PROGRAM TSCS_Bridge_Outputs
(*Outputs from TDU PLC to TSCS PLC*)
VAR
	// Function Blocks
	fb_Bridge_Outputs_Real_0 : FB_Bridge_Outputs_Real; // Interface for TDU real outputs
	
	// Signal Conversions
	rActPos : REAL; // Rotation system - Actual Position [deg]
	rActVel : REAL; // Rotation system - Actual Velocity [rpm]
	rSetVelRaw : REAL; //Rotation system - Velocity setpoint raw [rpm] 
	
END_VAR

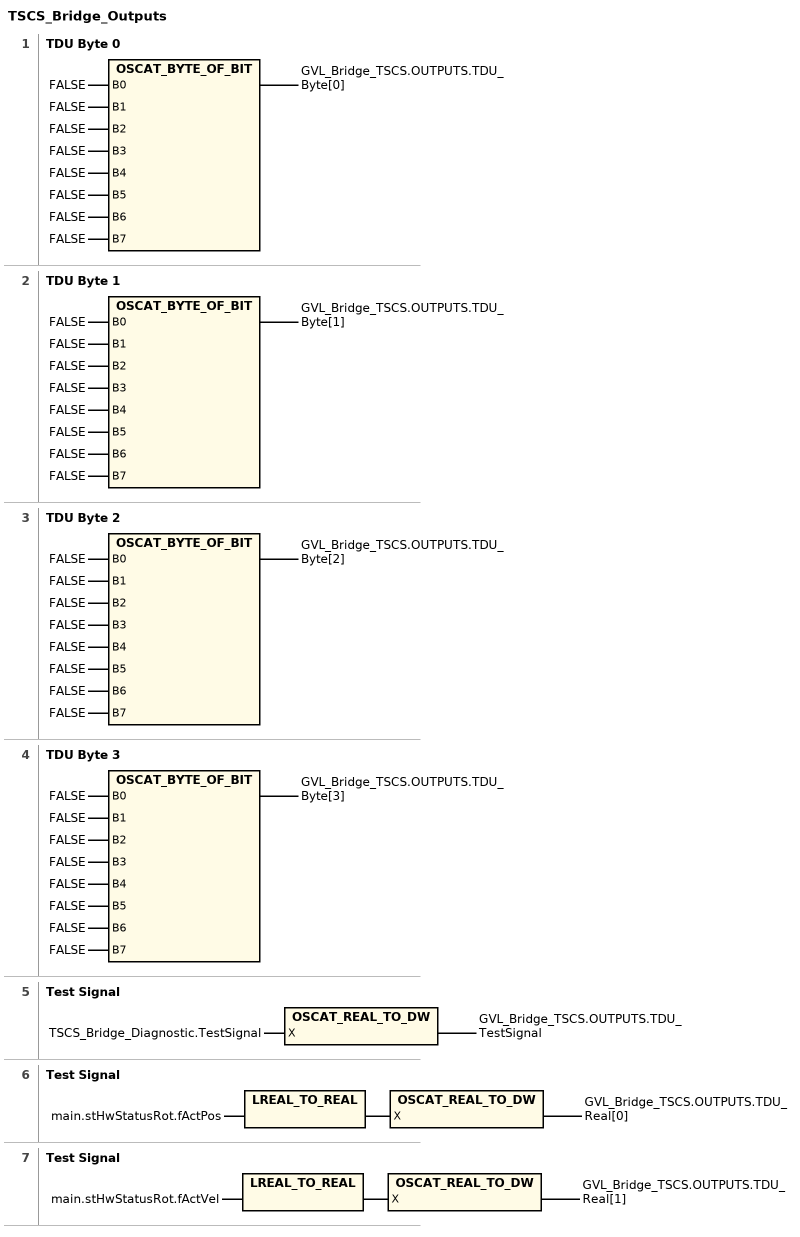
// NETWORK 1: TDU Byte 0
GVL_Bridge_TSCS.OUTPUTS.TDU_Byte[0] := OSCAT_BYTE_OF_BIT(B0 := FALSE, B1 := FALSE, B2 := FALSE, B3 := FALSE, B4 := FALSE, B5 := FALSE, B6 := FALSE, B7 := FALSE);

// NETWORK 2: TDU Byte 1
GVL_Bridge_TSCS.OUTPUTS.TDU_Byte[1] := OSCAT_BYTE_OF_BIT(B0 := FALSE, B1 := FALSE, B2 := FALSE, B3 := FALSE, B4 := FALSE, B5 := FALSE, B6 := FALSE, B7 := FALSE);

// NETWORK 3: TDU Byte 2
GVL_Bridge_TSCS.OUTPUTS.TDU_Byte[2] := OSCAT_BYTE_OF_BIT(B0 := FALSE, B1 := FALSE, B2 := FALSE, B3 := FALSE, B4 := FALSE, B5 := FALSE, B6 := FALSE, B7 := FALSE);

// NETWORK 4: TDU Byte 3
GVL_Bridge_TSCS.OUTPUTS.TDU_Byte[3] := OSCAT_BYTE_OF_BIT(B0 := FALSE, B1 := FALSE, B2 := FALSE, B3 := FALSE, B4 := FALSE, B5 := FALSE, B6 := FALSE, B7 := FALSE);

// NETWORK 5: Test Signal
GVL_Bridge_TSCS.OUTPUTS.TDU_TestSignal := OSCAT_REAL_TO_DW(X := TSCS_Bridge_Diagnostic.TestSignal);

// NETWORK 6: Test Signal
GVL_Bridge_TSCS.OUTPUTS.TDU_Real[0] := OSCAT_REAL_TO_DW(X := LREAL_TO_REAL(main.stHwStatusRot.fActPos));

// NETWORK 7: Test Signal
GVL_Bridge_TSCS.OUTPUTS.TDU_Real[1] := OSCAT_REAL_TO_DW(X := LREAL_TO_REAL(main.stHwStatusRot.fActVel));

END_PROGRAM

(* stored: Version 1.1.0.1, ProductVersion 3.1.4024.6
   POU TSCS_Bridge_Outputs: Id {3c6c9e4f-6ebc-4e74-8e61-0502fd6692d6}, SpecialFunc None *)
